(* Logix 5000 project; controller STAT 1756-L72 rev 20.12; software revision 20.04; part 31 of 34 *)
(* tags used below, declared in another part *)
   AUX_COND_KOELTOREN : REAL;
   AUX_LVL_KOEL : DINT;
   def_temp_iwts : BOOL;
   dmd_h2so4_ibt_ok : BOOL;
   ibtlancy1 : DINT;
   INT_COND_KOEL : integrat;
   INT_LVL_KOEL : integrat;
   L1_stat : DINT[20];
   L2_L3_OK : BOOL;
   L2_L3_ppas : DINT;
   L2_STAT : DINT[20];
   LVL_NITRIC : REAL;
   msg_W_lancy2 : MESSAGE;
   N : INT[255];
   naohL1VA4 : BOOL;
   naohL2VA4 : BOOL;
   op010 : DINT;
   real : REAL;
   S_BP_L2L3 : BOOL;
   S_COND_KOELTOREN : DINT;
   S_L2L3_Q_NAOH : DINT;
   S_LVL_KOELTOREN : DINT;
   S_LVL_nitric : REAL;
   S_STOCK_H2SO4 : DINT;
   S_STOCK_MAZ : DINT;
   S_STOCK_NAOH : DINT;
   S_T_CABINE_RED : DINT;
   S_T_in_CH_L3 : DINT;
   S_T_in_chaud_L123 : DINT;
   S_T_IWTS : DINT;
   S_T_OUT_CH_L3 : DINT;
   S_T_out_chaud_L123 : DINT;
   SCP_COND_KOELTOREN : SCP;
   SCP_LVL_KOELTOREN : SCP;
   SCP_lvl_nitric : SCP;
   scp_stck_acid : SCP;
   scp_stck_maz : SCP;
   scp_stck_soude : SCP;
   SCP_T_CABINE_L1 : SCP;
   scp_T_in_CH_L3 : SCP;
   scp_T_in_L12 : SCP;
   scp_T_iwts : SCP;
   scp_T_OUT_CH_L3 : SCP;
   scp_T_out_L12 : SCP;
   Seconde : BOOL;
   stat_L1 : DINT[20];
   stocklancy1 : DINT;
   stocklancy2 : DINT;
   stocklancy3 : DINT;
   stocklancy5 : DINT;   // alarme lvl 2 stock
   T1_cligno : TIMER;
   T_CABINE_RED : REAL;
   T_R_L2L3 : TIMER;
(* LANCY, continued *)

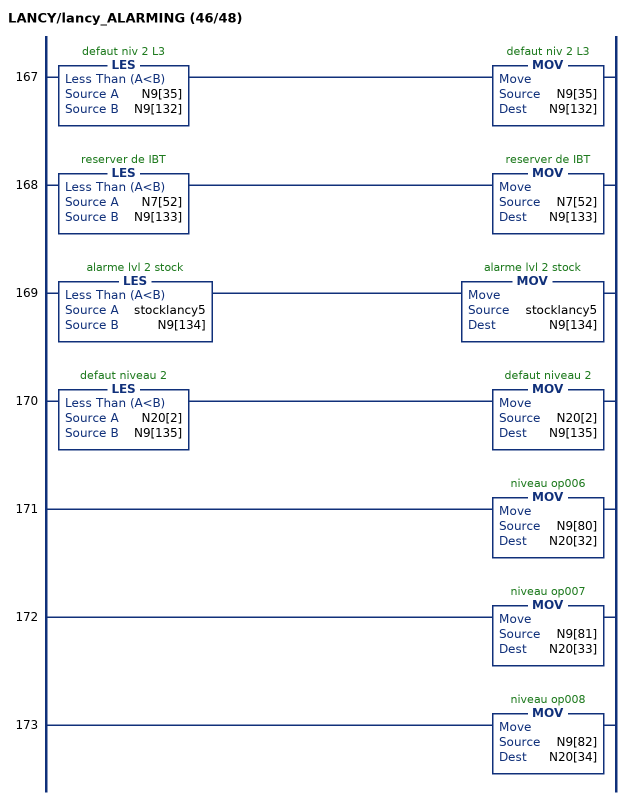
   [picture p626: LANCY/lancy_ALARMING rungs 167-173]
   167: LES(N9[35],N9[132])MOV(N9[35],N9[132]);
   168: LES(N7[52],N9[133])MOV(N7[52],N9[133]);
   169: LES(stocklancy5,N9[134])MOV(stocklancy5,N9[134]);
   170: LES(N20[2],N9[135])MOV(N20[2],N9[135]);
   171: MOV(N9[80],N20[32]);
   172: MOV(N9[81],N20[33]);
   173: MOV(N9[82],N20[34]);
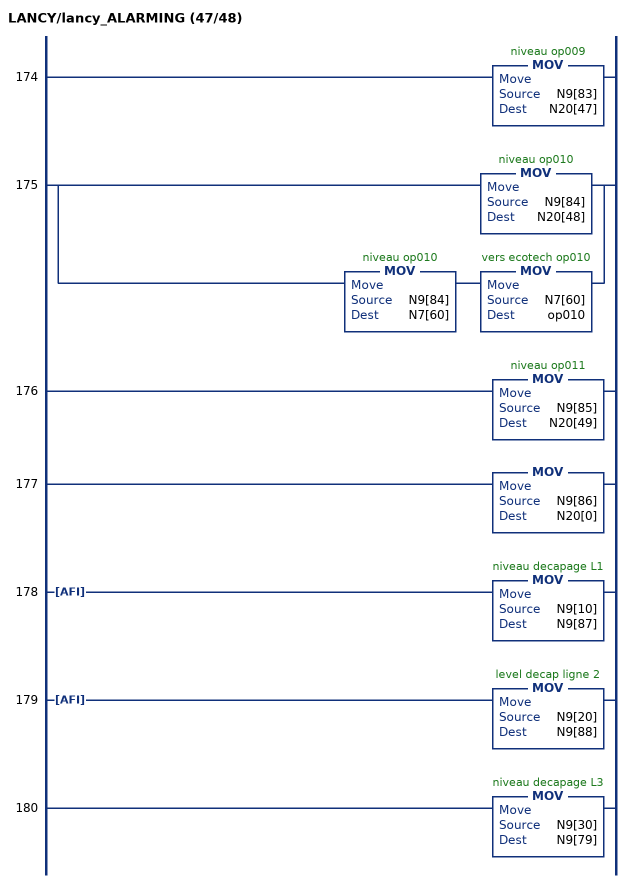
   174: MOV(N9[83],N20[47]);
   175: [MOV(N9[84],N20[48]) ,MOV(N9[84],N7[60]) MOV(N7[60],op010) ];
   176: MOV(N9[85],N20[49]);
   177: MOV(N9[86],N20[0]);
   178: AFI()MOV(N9[10],N9[87]);
   179: AFI()MOV(N9[20],N9[88]);
   180: MOV(N9[30],N9[79]);
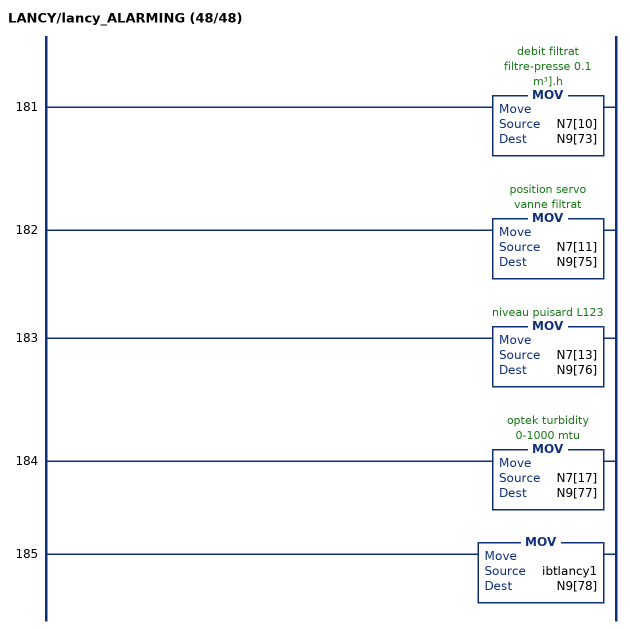
   181: MOV(N7[10],N9[73]);
   182: MOV(N7[11],N9[75]);
   183: MOV(N7[13],N9[76]);
   184: MOV(N7[17],N9[77]);
   185: MOV(ibtlancy1,N9[78]);
END_ROUTINE

ROUTINE lancy_apport_soude   (* ladder *)
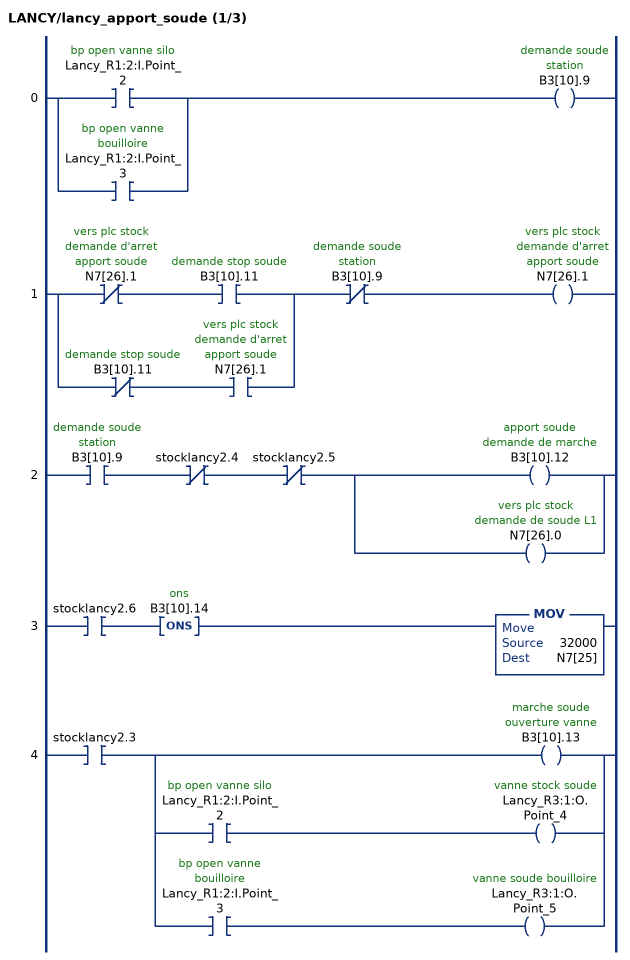
   0: [XIC(Lancy_R1:2:I.Point_2) ,XIC(Lancy_R1:2:I.Point_3) ]OTE(B3[10].9);
   1: [XIO(N7[26].1) XIC(B3[10].11) ,XIO(B3[10].11) XIC(N7[26].1) ]XIO(B3[10].9)OTE(N7[26].1);
   2: XIC(B3[10].9)XIO(stocklancy2.4)XIO(stocklancy2.5)[OTE(B3[10].12) ,OTE(N7[26].0) ];
   3: XIC(stocklancy2.6)ONS(B3[10].14)MOV(32000,N7[25]);
   4: XIC(stocklancy2.3)[OTE(B3[10].13) ,XIC(Lancy_R1:2:I.Point_2) OTE(Lancy_R3:1:O.Point_4) ,XIC(Lancy_R1:2:I.Point_3) OTE(Lancy_R3:1:O.Point_5) ];
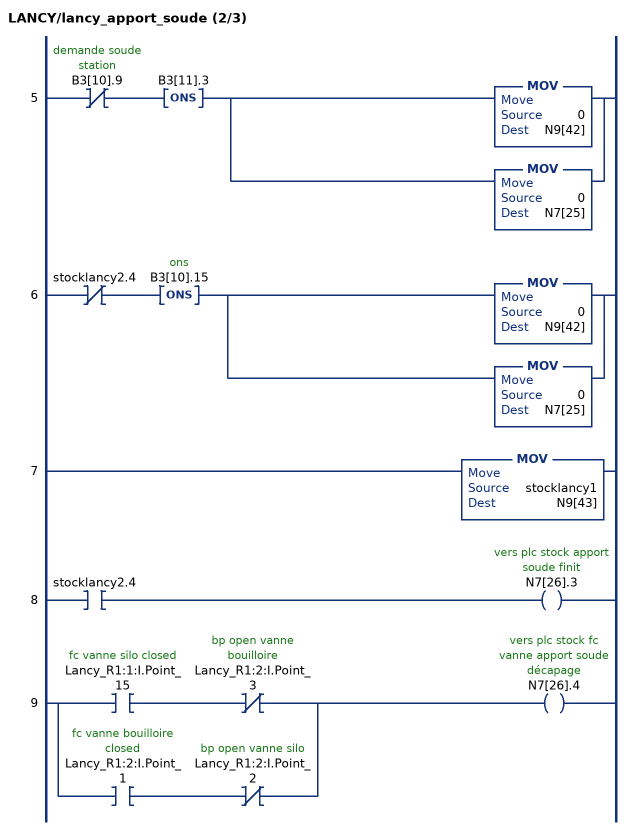
   5: XIO(B3[10].9)ONS(B3[11].3)[MOV(0,N9[42]) ,MOV(0,N7[25]) ];
   6: XIO(stocklancy2.4)ONS(B3[10].15)[MOV(0,N9[42]) ,MOV(0,N7[25]) ];
   7: MOV(stocklancy1,N9[43]);
   8: XIC(stocklancy2.4)OTE(N7[26].3);
   9: [XIC(Lancy_R1:1:I.Point_15) XIO(Lancy_R1:2:I.Point_3) ,XIC(Lancy_R1:2:I.Point_1) XIO(Lancy_R1:2:I.Point_2) ]OTE(N7[26].4);
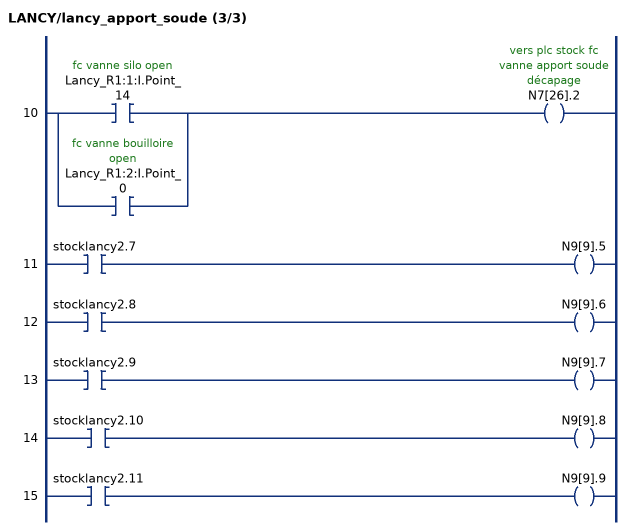
   10: [XIC(Lancy_R1:1:I.Point_14) ,XIC(Lancy_R1:2:I.Point_0) ]OTE(N7[26].2);
   11: XIC(stocklancy2.7)OTE(N9[9].5);
   12: XIC(stocklancy2.8)OTE(N9[9].6);
   13: XIC(stocklancy2.9)OTE(N9[9].7);
   14: XIC(stocklancy2.10)OTE(N9[9].8);
   15: XIC(stocklancy2.11)OTE(N9[9].9);
END_ROUTINE

ROUTINE NAOH   (* ladder *)
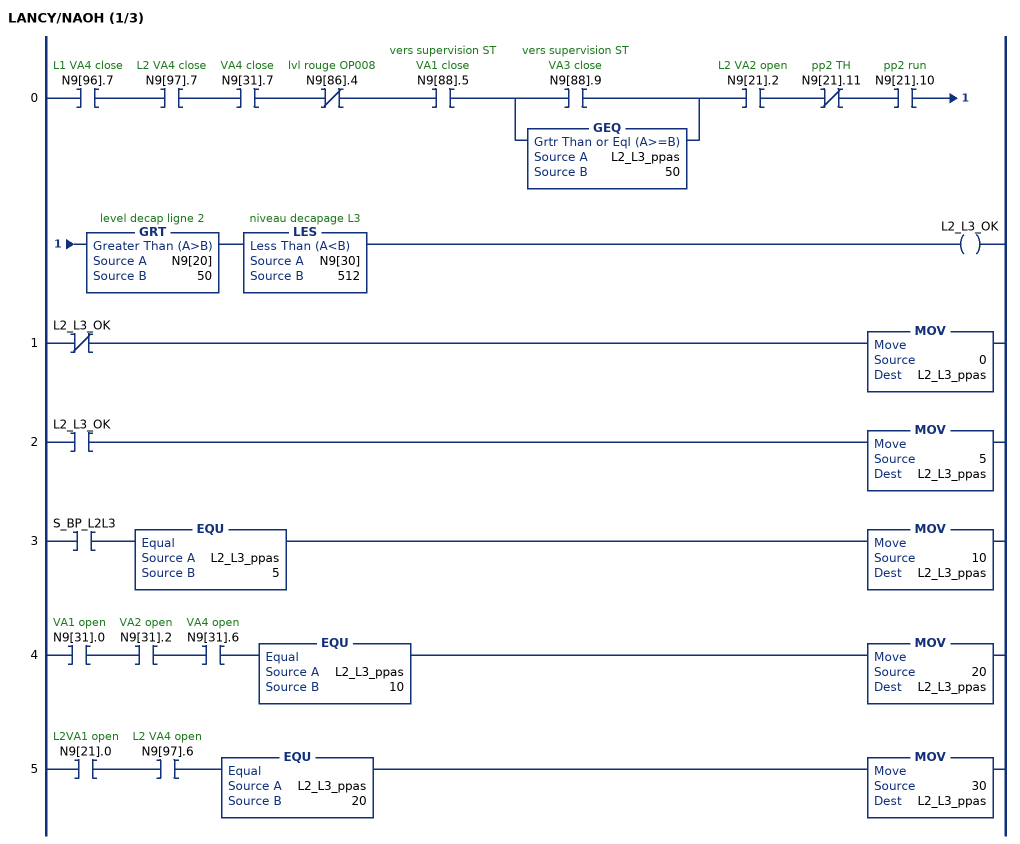
   0: XIC(N9[96].7)XIC(N9[97].7)XIC(N9[31].7)XIO(N9[86].4)XIC(N9[88].5)[XIC(N9[88].9) ,GEQ(L2_L3_ppas,50) ]XIC(N9[21].2)XIO(N9[21].11)XIC(N9[21].10)GRT(N9[20],50)LES(N9[30],512)OTE(L2_L3_OK);
   1: XIO(L2_L3_OK)MOV(0,L2_L3_ppas);
   2: XIC(L2_L3_OK)MOV(5,L2_L3_ppas);
   3: XIC(S_BP_L2L3)EQU(L2_L3_ppas,5)MOV(10,L2_L3_ppas);
   4: XIC(N9[31].0)XIC(N9[31].2)XIC(N9[31].6)EQU(L2_L3_ppas,10)MOV(20,L2_L3_ppas);
   5: XIC(N9[21].0)XIC(N9[97].6)EQU(L2_L3_ppas,20)MOV(30,L2_L3_ppas);
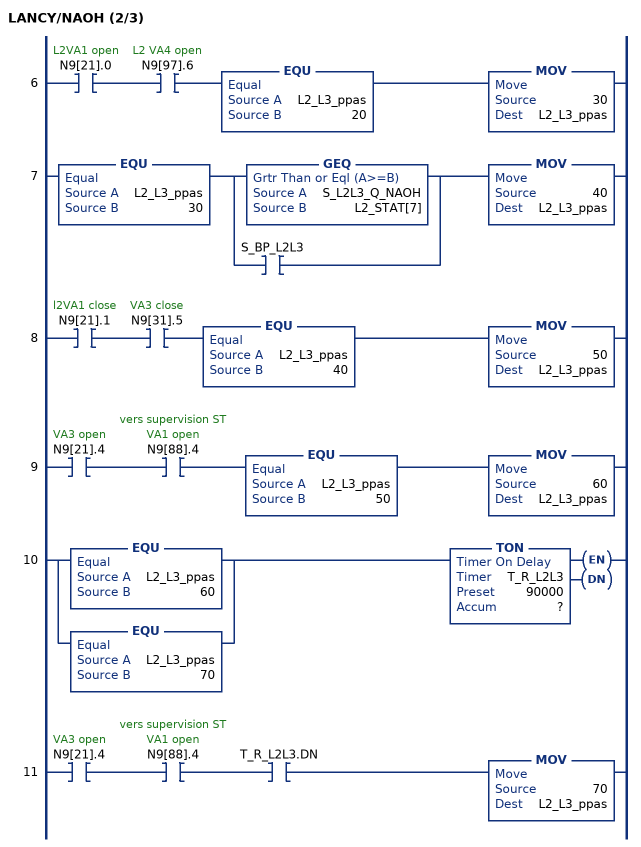
   6: XIC(N9[21].0)XIC(N9[97].6)EQU(L2_L3_ppas,20)MOV(30,L2_L3_ppas);
   7: EQU(L2_L3_ppas,30)[GEQ(S_L2L3_Q_NAOH,L2_STAT[7]) ,XIC(S_BP_L2L3) ]MOV(40,L2_L3_ppas);
   8: XIC(N9[21].1)XIC(N9[31].5)EQU(L2_L3_ppas,40)MOV(50,L2_L3_ppas);
   9: XIC(N9[21].4)XIC(N9[88].4)EQU(L2_L3_ppas,50)MOV(60,L2_L3_ppas);
   10: [EQU(L2_L3_ppas,60) ,EQU(L2_L3_ppas,70) ]TON(T_R_L2L3,?,?);
   11: XIC(N9[21].4)XIC(N9[88].4)XIC(T_R_L2L3.DN)MOV(70,L2_L3_ppas);
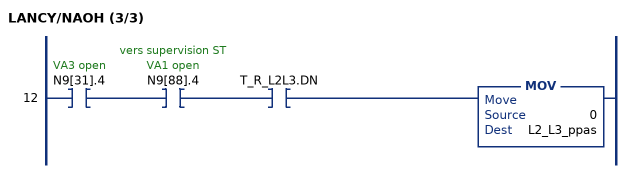
   12: XIC(N9[31].4)XIC(N9[88].4)XIC(T_R_L2L3.DN)MOV(0,L2_L3_ppas);
END_ROUTINE
END_PROGRAM

PROGRAM MainProgram
END_PROGRAM

PROGRAM stock   (* main routine MAIN_STOCK *)
VAR
   aa : DINT;
   B3 : DINT[50] := ([0] := 2#0000_0000_0000_0000_0000_1000_0010_0000, [2] := 2#0000_0000_0000_0000_0100_0010_1110_0000, [3] := 2#0000_0000_0000_0000_0000_0000_0000_0101, [5] := 2#0000_0000_0000_0000_0000_0000_1000_0000);
        [4].1   // L1 hs
        [4].2   // l2 hs
        [4].3   // l3 hs
        [0].0   // UNE VANNE SOUDE OUVERTE
        [0].4   // vanne acidedemarrage pompe
        [0].5   // one shot
        [0].6   // ons
        [0].7   // soude occupée
        [0].8   // soude déjaoccupé
        [0].9   // défautvanne soude
        [0].10   // ACIDE DEJAACCUPE
        [0].11   // ons
        [0].12   // acide occupe
        [0].14   // défautvanne acide
        [0].15   // AUX D2FAUTVANNE ACIDE
        [1].1   // ons
        [1].2   // apport soude
        [1].3   // acquit klaxonfuite acide
        [1].4   // acquit klaxonfuite soude
        [1].5   // acquit klaxonfuite mazout
        [1].6   // detectionfuiteacide
        [1].12   // apport acide
        [2].0   // ons
        [2].1   // ons
        [2].2   // ons
        [2].3   // ons
        [2].4   // ons
        [2].5   // ons
        [2].7   // ons
        [2].8   // ons
        [2].9   // ons
        [2].10   // ons
        [2].11   // ons
        [2].12   // ons
        [2].13   // ons
        [2].14   // ons
        [2].15   // ons
        [3].0   // fonctionnementdepuis supervision
        [3].1   // ARRET ENTRETIEN
        [3].2   // nouveau def
        [3].3   // rappel demandé
        [4].0   // stat hs
        [4].4   // l4 hs
        [5].7   // ons
   C5 : COUNTER[10];
   F8 : REAL[200] := ([2] := 863724.06, [3] := 863678.3, [5] := 24000.0, [7] := 1000.0, [10] := 17654.0, [11] := 20000.0, [12] := 9201.893, [13] := 48000.0, [14] := 24840.227, [15] := 45000.0, [16] := -750.11444, [17] := -750.11444, [18] := 2135.205, [19] := 2142.53, [20] := 2033.7975, [21] := 1750.6666, [22] := 2993.7632, [23] := 150.19885, [25] := 44558.395, [26] := 80344.15, [27] := 2182.817, [29] := 281.0, [30] := 24832.748, [31] := -3.7382812, [32] := 17654.0, [34] := 9201.893, [35] := -3.8154297, [36] := 5102.8765, [37] := 2410.5056, [38] := 7013.7407, [41] := 0.6, [42] := 50.0, [43] := 50.000046, [46] := -863724.06, [47] := 50.0, [48] := 50.000046, [50] := 318801.06, [52] := -318801.06, [61] := 1750.6666, [62] := 2993.7632, [63] := 150.19885);
        [2]   // 0.2 L].pulsetotalacide
        [3]   // memo acidepassé
        [4]   // quantitédernièreenvoi acide
        [10]   // Stock acide
        [12]   // stock mazout
        [14]   // stock soude
        [16]   // temperature entréeChaudière Ligne 1-2
        [17]   // temperature desortie chaudièreLigne 1-2
        [18]   // temp entréechaudierecolmatage L3
        [19]   // temp sortiechaudierecolmatage L3
        [20]   // total soudevers station
        [21]   // total soudevers L1
        [22]   // total soudevers L2
        [23]   // total soudevers L3
        [24]   // total soudevers L4
        [25]   // total soudevers L2
        [26]   // total soudevers L1
        [27]   // chaudiere iwts
        [30]   // NIVEAU PRECEDENTSOUDE
        [31]   // PERTE SOUDE SUR UNEMINUTE
        [32]   // PERTE ACIDE SUR UNEMIN
        [33]   // MEMO NIVEAI ACIDE1 MIN AVANT
        [34]   // MEMO MAZOUT 1 MIN
        [35]   // PERTE MAZOUT SUR1 MIN
        [36]   // totalacideL1
        [37]   // totalacideL2
        [38]   // totalacideL3
        [39]   // totalacideL4
        [40]   // quantité demandéedepuis ligne
        [41]   // quantité soudepassée
        [42]   // quantité acidedemandéedepuis ligne
        [43]   // quantité acidepassée
        [45]   // aux total acide
        [46]   // aux total acide
        [47]   // aux total acide
        [48]   // quantité acidepassé
        [50]   // total soudepassée en L
        [62]   // MEMO FLOW TO L2
        [63]   // MEMO FLOW TO L3
   I1 : DINT;
   I1_000_Bit00 : ALIAS FOR stock:1:I.Point_0;   // disjoncteur algemeen
   I1_000_Bit01 : ALIAS FOR stock:1:I.Point_1;   // alim rechauffeur1
   I1_000_Bit02 : ALIAS FOR stock:1:I.Point_2;   // alim rechauffeur2
   I1_000_Bit03 : ALIAS FOR stock:1:I.Point_3;   // alim rechauffeur 3
   I1_000_Bit04 : ALIAS FOR stock:1:I.Point_4;   // alim rechauffeur 4
   I1_000_Bit05 : ALIAS FOR stock:1:I.Point_5;   // alim rechauffeur 5
   I1_000_Bit06 : ALIAS FOR stock:1:I.Point_6;   // protection pompesoude
   I1_000_Bit07 : ALIAS FOR stock:1:I.Point_7;   // protection pmp 2 acide
   I1_000_Bit08 : ALIAS FOR stock:1:I.Point_8;   // protection pmp acide
   I1_000_Bit09 : ALIAS FOR stock:1:I.Point_9;
   I1_000_Bit10 : ALIAS FOR stock:1:I.Point_10;
   I1_000_Bit11 : ALIAS FOR stock:1:I.Point_11;
   I1_000_Bit12 : ALIAS FOR stock:1:I.Point_12;
   I1_000_Bit15 : ALIAS FOR stock:1:I.Point_15;   // arret urgence
   I1_001_Bit01 : ALIAS FOR stock:1:I.Point_17;   // reset arret urgence
   I1_001_Bit02 : ALIAS FOR stock:1:I.Point_18;   // start pompe soude
   I1_001_Bit03 : ALIAS FOR stock:1:I.Point_19;   // stop pompe soude
   I1_001_Bit04 : ALIAS FOR stock:1:I.Point_20;   // start pompe acide
   I1_001_Bit05 : ALIAS FOR stock:1:I.Point_21;   // stop pompe acide
   I1_001_Bit08 : ALIAS FOR stock:1:I.Point_24;   // local ]. distance
   I1_001_Bit09 : ALIAS FOR stock:1:I.Point_25;   // select.pmp soude sur drive
   I1_001_Bit10 : ALIAS FOR stock:1:I.Point_26;   // select.pmp soude sur ultima
   I1_001_Bit11 : ALIAS FOR stock:1:I.Point_27;   // fault drivepmp soude
   I2 : DINT;
   I2_000_Bit00 : ALIAS FOR stock:2:I.Point_0;   // detection fuite soud
   I2_000_Bit01 : ALIAS FOR stock:2:I.Point_1;   // detection fuite acid
   I2_000_Bit02 : ALIAS FOR stock:2:I.Point_2;   // detection fuite mazo
   I2_000_Bit03 : ALIAS FOR stock:2:I.Point_3;   // wegskraan soude open
   I2_000_Bit04 : ALIAS FOR stock:2:I.Point_4;   // wegskraan soude dich
   I2_000_Bit05 : ALIAS FOR stock:2:I.Point_5;   // start pompe acidedepuis ligne
   I2_000_Bit06 : ALIAS FOR stock:2:I.Point_6;   // start pompe acidedepuis ligne RESERVE
   I2_000_Bit07 : ALIAS FOR stock:2:I.Point_7;   // overfill stockagesoude
   I2_000_Bit08 : ALIAS FOR stock:2:I.Point_8;   // detection acideencuvement
   I2_000_Bit09 : ALIAS FOR stock:2:I.Point_9;   // detection soudeencuvement
   I2_000_Bit10 : ALIAS FOR stock:2:I.Point_10;   // fv vannesecuriteacide OUVERT
   I2_000_Bit11 : ALIAS FOR stock:2:I.Point_11;   // fv vannesecuriteacide FERME
   I2_000_Bit12 : ALIAS FOR stock:2:I.Point_12;   // chaudière wanson0= on 1= off
   I2_000_Bit13 : ALIAS FOR stock:2:I.Point_13;   // chaudière colmatageLigne 30= on 1= off
   I2_000_Bit14 : ALIAS FOR stock:2:I.Point_14;   // DEFAUT CHAUDIEREiwts
   I2_001_Bit00 : ALIAS FOR stock:2:I.Point_16;   // NAOHL1 VA4FC O
   I2_001_Bit01 : ALIAS FOR stock:2:I.Point_17;   // NAOHL1 VA4FC F
   I2_001_Bit02 : ALIAS FOR stock:2:I.Point_18;   // NAOHL2 VA4FC O
   I2_001_Bit03 : ALIAS FOR stock:2:I.Point_19;   // NAOHL2 VA4FC O
   I2_001_Bit06 : ALIAS FOR stock:2:I.Point_22;   // pulse debitmetreacide 0.2 l
   I2_001_Bit07 : ALIAS FOR stock:2:I.Point_23;   // pulse eau in tourL1 &2
   I2_001_Bit15 : ALIAS FOR stock:2:I.Point_31;   // pulse 0.1L passé
   I4 : AB:1746_NI8_C63AF0D1:I:0;
   I4_001 : ALIAS FOR stock:4:I.Channel_1_Data;   // level soude
   I4_002 : ALIAS FOR stock:4:I.Channel_2_Data;   // level acide
   I4_003 : ALIAS FOR stock:4:I.Channel_3_Data;   // level mazout
   I4_004 : ALIAS FOR stock:4:I.Channel_4_Data;
   I4_005 : ALIAS FOR stock:4:I.Channel_5_Data;
   I4_006 : ALIAS FOR stock:4:I.Channel_6_Data;
   I4_007 : ALIAS FOR stock:4:I.Channel_7_Data;
   I5 : INT[8] := ([0] := 2#0000_1100_1100_1101, [1] := 2#0001_0000_0011_0101, [2] := 2#0011_0111_1011_0100, [3] := 2#0001_0001_1111_1000, [4] := 2#0000_1100_1101_0101, [5] := 2#0001_1000_1001_0100);
   I5_000 : ALIAS FOR stock:5:I.Channel_0_Data;
   I5_001 : ALIAS FOR stock:5:I.Channel_1_Data;
   I5_002 : ALIAS FOR stock:5:I.Channel_2_Data;
   I5_003 : ALIAS FOR stock:5:I.Channel_3_Data;
   I5_004 : ALIAS FOR stock:5:I.Channel_4_Data;
   I5_005 : ALIAS FOR stock:5:I.Channel_5_Data;
   N20 : DINT[100] := ([1] := 8, [2] := 3, [5] := 3, [10] := 2, [20] := 64, [21] := 61967, [25] := 64, [30] := 10, [31] := 1);
        [1]   // DEFAUT PRIORITE 1
        [2]   // DEFAUT PRIORITE 2
        [5].0   // DEFAULT
        [5].1   // NEW DEFAULT
        [9].1   // ack STOCK
        [10].0   // chaudiere wanson on
        [10].1   // chaudière colmatageLigne 3 on
        [20].0   // defautdisjoncteur algemeen
        [20].1   // DEFAUTalim rechauffeur1
        [20].2   // DEFAUTalim rechauffeur2
        [20].3   // DEFAUTalim rechauffeur 3
        [20].4   // DEFAUTalim rechauffeur 4
        [20].5   // DEFAUTalim rechauffeur 5
        [20].6   // DEFAUTprotection pompesoude
        [20].7   // DEFAUTprotection pmpmazout
        [20].8   // DEFAUTprotection pmp acide
        [20].9   // DEFAUTarret urgence
        [20].10   // DEFAUTdetection fuite soud
        [20].11   // DEFAUTdetection fuite acid
        [20].12   // DEFAUTdetection fuite mazo
        [20].13   // DEFAUToverfill stockagesoude
        [20].14   // DEFAUTdetection acideencuvement
        [20].15   // DEFAUTdetection soudeencuvement
        [21].0   // DEFAUTPOSITION VANNEL1 VA4
        [21].1   // DEFAUTPOSITION VANNEL2 VA4
        [21].2   // DEFAUTPOSITION VANNESOUDE VERS LIGNES
        [21].3   // DEFAUTPOSITION VANNEACIDE VERS LIGNES
        [21].4   // DEFAUT FLOW SOUDE
        [21].5   // DEFAUT NIVEAU SOUDEHH
        [21].6   // DEFAUT NIVEAU SOUDELL
        [21].7   // DEFAUT FILL OUTNOAH TANK
        [21].8   // DEFAUT NIVEAU ACIDEHH
        [21].9   // DEFAUT NIVEAU ACIDELL
        [21].10   // DEFAUT FILL OUTH2SO4 TANK
        [21].11   // DEFAUT NIVEAU MAZOUTHH
        [21].12   // DEFAUT NIVEAU MAZOUTLL
        [21].13   // DEFAUT FILL OUTMAZOUT TANK
        [21].14   // DEFAUT CHAUDIEREiwts
        [21].15   // defautchaudierecolmatage L3
        [25].0   // defautdisjoncteur algemeen
        [25].1   // DEFAUTalim rechauffeur1
        [25].2   // DEFAUTalim rechauffeur2
        [25].3   // DEFAUTalim rechauffeur 3
        [25].4   // DEFAUTalim rechauffeur 4
        [25].5   // DEFAUTalim rechauffeur 5
        [25].6   // DEFAUTprotection pompesoude
        [25].7   // DEFAUTprotection pmpmazout
        [25].8   // DEFAUTprotection pmp acide
        [25].9   // DEFAUTarret urgence
        [25].10   // DEFAUTdetection fuite soud
        [25].11   // DEFAUTdetection fuite acid
        [25].12   // DEFAUTdetection fuite mazo
        [25].13   // overfill stockagesoude
        [25].14   // DEFAUTdetection acideencuvement
        [25].15   // DEFAUTdetection soudeencuvement
        [26].0   // DEFAUTPOSITION VANNEL1 VA4
        [26].1   // DEFAUTPOSITION VANNEL2 VA4
        [26].2   // DEFAUTPOSITION VANNESOUDE VERS LIGNES
        [26].3   // DEFAUTPOSITION VANNEACIDE VERS LIGNES
        [26].4   // DEFAUT FLOW SOUDE
        [26].5   // DEFAUT NIVEAU SOUDEHH
        [26].6   // DEFAUT NIVEAU SOUDELL
        [26].7   // DEFAUT FILL OUTNOAH TANK
        [26].8   // DEFAUT NIVEAU ACIDEHH
        [26].9   // DEFAUT NIVEAU ACIDELL
        [26].10   // DEFAUT FILL OUTH2SO4 TANK
        [26].11   // DEFAUT NIVEAU MAZOUTHH
        [26].12   // DEFAUT NIVEAU MAZOUTLL
        [26].13   // DEFAUT FILL OUTMAZOUT TANK
        [26].14   // DEFAUT CHAUDIEREiwts
        [26].15   // memo defautchaudierecolmatage L3
        [30]   // NOMBRE DE DEFAUTS
        [31]   // MEMONOMBRE DE DEFAUTS
   N7 : DINT[255] := ([1] := 131701, [3] := 3850, [4] := 3800, [10] := 21, [15] := 281, [18] := 314857, [20] := 10, [21] := -4, [66] := -32752, [68] := 336, [88] := 50, [108] := 80, [126] := 3488, [127] := 35200, [166] := 3488, [167] := 35200, [206] := 3488, [207] := 35200, [246] := 3488);
        [1]   // gxf
        [2]   // flow acide
        [10].0   // stock acide pas haut
        [10].1   // stock acide pas bas
        [10].2   // stock mazout pashaut
        [10].3   // stock mazout pas bas
        [10].4   // stock soude L1 pashaut
        [10].5   // stock soude L1 pasbas
        [10].7   // stock soude L2 pasbas
        [10].8   // stock soude L3 pashaut
        [10].9   // stock soude L3 pasbas
        [10].10   // PVvanne soude L1fermée
        [10].13   // de PVchargement en cours
        [10].14   // DE PVBP EV SOUDE L1
        [11].0   // DE PVBP EV SOUDE L3
        [11].1   // vers PVfuite stock acide
        [11].2   // vers PVfuite stock mazout
        [11].3   // fuite soude
        [15]   // T° ambiantecabine RED L1
        [16]   // conductivité en µS
        [17]   // niveau eautour refroidissement
        [18]   // total eau tour L1 2
        [20].0   // NAOHL1 VA4FC O
        [20].1   // NAOHL1 VA4FC F
        [20].2   // NAOHL2 VA4FC O
        [20].3   // NAOHL2 VA4FC F
        [30]   // MESSAGE TO LANCY
        [46].2   // DE PLC 1VANNE SOUDEL1 OUVERTE
        [50]   // communication avecplc L1 read
        [65]   // quantité soudedemandée L1
        [66].0   // DE PLC L1demande soudeL1
        [66].1   // DE PLC L1demandearret soude L1
        [66].2   // de plc ligne 1fc vanne soudeouverte
        [66].3   // de plc ligne 1apport soudefinit
        [66].4   // de plc ligne 1fc vanne soudefermée
        [66].15   // de line 1line 1 run
        [67]   // quantité acidedemandée L1
        [68].0   // DE PLC L1demande acide
        [68].1   // DE PLC L1demandearret acide L1
        [68].2   // de plc ligne 1fc vanne acideano ouv
        [68].3   // de plc ligne 1apport acidefinit
        [68].4   // de plc ligne 1fc vanne acideano ferme
        [68].5   // de plc ligne 1fc vanne acideneut ouv
        [68].6   // de plc ligne 1fc vanne acideneut ferme
        [68].7   // de plc ligne 1fc vanne acidecolo ouv
        [68].8   // de plc ligne 1fc vanne acidecolo fermé
        [70]   // communication avecplc L1 write
        [85]   // quantité souderestante L1
        [86].0   // vers plc l1 fuiteacide
        [86].1   // vers plc l1fuite soude
        [86].2   // vers plc L1fuite mazout
        [86].3   // vers plc L1ouvrir vannesoude
        [86].4   // vers plc L1apport soudefinit L1
        [86].5   // vers plc L1apport soudeoccupé
        [86].6   // vers plc L1apport soudeL1 accordé
        [86].7   // VERS PLC L1SOUDE VERS L1
        [86].8   // VERS PLC L1SOUDE VERS L2
        [86].9   // VERS PLC L1SOUDE VERS L3
        [86].10   // VERS PLC L1SOUDE VERS L4
        [86].11   // VERS PLC L1SOUDE VERS STAT
        [86].12   // DEFAULT FLOW TO L1VERS SLC
        [87]   // vers plc L1
        [87].3   // vers plc L1ouvrir vanneacide
        [87].4   // vers plc L1apport acidefinit L1
        [87].5   // vers plc L1apport acideoccupé
        [87].6   // vers plc L1apport acideaccordé
        [87].7   // VERS PLC L1acide VERS ano L1
        [87].8   // VERS PLC L1acideVERS L2
        [87].9   // VERS PLC L1acide VERS L3
        [87].10   // VERS PLC L1acide VERS L4
        [87].11   // VERS PLC L1acide VERS neutralL1
        [87].12   // VERS PLC L1 acideneutralL2
        [87].13   // VERS PLC L1acide neutralL3
        [87].14   // VERS PLC L1 acide VEL4
        [88]   // quantité aciderestante L1
        [90]   // communication avecplc L2 read
        [105]   // quantité soudedemandée L2
        [106].0   // DE PLC L2demande soudeL2
        [106].1   // DE PLC L2demandearret soude
        [106].2   // de plc ligne 2fc vanne soudeouverte
        [106].4   // de plc ligne 2fc vanne soudefermée
        [106].15   // de line 2line 2 run
        [107]   // quantité acidedemandée L2
        [108].0   // DE PLC L2demande acide
        [108].1   // DE PLC L2demandearret acide L2
        [108].2   // de plc ligne 2fc vanne acideouverte
        [108].4   // de plc ligne 2fc vanne acidefermée
        [108].5   // de plc ligne 2fc vanne acideneutral ouv
        [108].6   // de plc ligne 2fc vanne acideneutral ferm
        [110]   // communication avecplc L2 write
        [125]   // quantité souderestante L2
        [126].3   // vers plc L2ouvrir vannesoude
        [126].4   // vers plc L2apport soudefinit L2
        [126].5   // vers plc L2apport soudeoccupé
        [126].6   // vers plc L2apport soudeL2 accordé
        [126].7   // VERS PLC L2SOUDE VERS L1
        [126].8   // VERS PLC L2SOUDE VERS L2
        [126].9   // VERS PLC L2SOUDE VERS L3
        [126].10   // VERS PLC L2SOUDE VERS L4
        [126].11   // VERS PLC L2SOUDE VERS STAT
        [126].12   // DEFAULT FLOW TO L2VERS SLC
        [127].3   // vers plc L2ouvrir vanneacide
        [127].4   // vers plc L2apport acidefinit L2
        [127].5   // vers plc L2apport acideoccupé
        [127].6   // vers plc L2apport acideaccordé
        [127].7   // VERS PLC L2acide VERS ano L1
        [127].8   // VERS PLC L2acide VERS L2
        [127].9   // VERS PLC L2acide VERS L3
        [127].10   // VERS PLC L2acide VERS L4
        [127].11   // VERS PLC L2acide VERS neutralL1
        [127].12   // VERS PLC L2 acideneutralL2
        [127].13   // VERS PLC L2 acideneutralL3
        [127].14   // VERS PLC L2 acide VEL4
        [128]   // quantite acidepassé l2
        [130]   // communication L3read
        [139]   // MEMODEFAUT DEGRAISSAGE
        [145]   // quantité soudedemandéel3
        [146].0   // DE PLC L3demande soudeL3
        [146].1   // DE PLC L3demandearret soude L3
        [146].2   // de plc ligne 3fc vanne soudeouverte
        [146].4   // de plc ligne 3fc vanne soudefermée
        [146].15   // ligne 3 runcolmatage
        [147]   // quantité acidedemandée l3
        [148].0   // DE PLC L3demande acide L3
        [148].1   // DE PLC L3demandearret acide L3
        [148].2   // de plc ligne 3fc vanneacide ouverte
        [148].4   // de plc ligne 3fc vanne acidefermée
        [148].5   // de plc ligne 3fc vanneacide neutral ouv
        [148].6   // de plc ligne 3fc vanneacide neutral ferm
        [150]   // communication L3write
        [165]   // quantité souderestante L3
        [166].3   // vers plc L3ouvrir vannesoude
        [166].4   // vers plc L3apport soudeL3 finit
        [166].5   // vers plc L3apport soudeoccupé
        [166].6   // vers plc L3apport soudeL3 accordé
        [166].7   // VERS PLC L3SOUDE VERS L1
        [166].8   // VERS PLC L3SOUDE VERS L2
        [166].9   // VERS PLC L3SOUDE VERS L3
        [166].10   // VERS PLC L3SOUDE VERS L4
        [166].11   // VERS PLC L3SOUDE VERS STAT
        [166].12   // DEFAULT FLOW TO L3VERS SLC
        [167].3   // vers plc L3ouvrir vanneacide
        [167].4   // vers plc L3apport acidefinit L3
        [167].5   // apport acide occupé
        [167].6   // apport acide accordé
        [167].7   // VERS PLC L3acide VERS ano L1
        [167].8   // VERS PLC L3acide VERS L2
        [167].9   // VERS PLC L3acide VERS L3
        [167].10   // VERS PLC L4acide VERS L4
        [167].11   // VERS PLC L3acide VERS neutralL1
        [167].12   // VERS PLC L3 acideneutralL2
        [167].13   // VERS PLC L3acideneutral L3
        [167].14   // VERS PLC L3 acide VEL4
        [168]   // quantite acidepassé l3
        [170]   // communicationL4
        [185]   // quantité soudedemandéel4
        [186].0   // DE PLC L4demande soudeL4
        [186].1   // DE PLC L4demandearret soude l4
        [186].2   // de plc ligne 4fc vanne soudeouverte
        [186].4   // de plc ligne 4fc vanne soudefermée
        [187]   // quantité acidedemandée L4
        [188].0   // DE PLC L4demande acide
        [188].1   // DE PLC L4demandearret acide L4
        [188].2   // de plc ligne 4fc vanne acideouverte
        [188].4   // de plc ligne 3fc vanne acidefermée
        [188].5   // de plc ligne 4fc vanne acideneutral ouv
        [188].6   // de plc ligne 4fc vanne acideneutral ferme
        [190]   // communicationL4
        [205]   // quantité souderestante L4
        [206].3   // vers plc L4ouvrir vannesoude
        [206].4   // vers plc L4apport soudeL4 finit
        [206].5   // vers plc L4apport soudeoccupé
        [206].6   // vers plc L4apport soudeL4 accordé
        [206].7   // VERS PLC L4SOUDE VERS L1
        [206].8   // VERS PLC L4SOUDE VERS L2
        [206].9   // VERS PLC L4SOUDE VERS L3
        [206].10   // VERS PLC L4SOUDE VERS L4
        [206].11   // VERS PLC L4SOUDE VERS STAT
        [207].3   // vers plc L4ouvrir vanneacide
        [207].4   // vers plc L4apport acidefinit L4
        [207].5   // vers plc L4apport acideoccupé
        [207].6   // vers plc L4apport acideaccordé
        [207].7   // VERS PLC L4acide VERS ano L1
        [207].8   // VERS PLC L4acide VERS L2
        [207].9   // VERS PLC L4acide VERS L3
        [207].10   // VERS PLC L4acide VERS L4
        [207].11   // VERS PLC L4acide VERS neutralL1
        [207].12   // VERS PLC L4 acideneutralL2
        [207].13   // VERS PLC L4acide neutralL3
        [207].14   // VERS PLC L4 acide VEL4
        [208]   // quantite acidepassé l4
        [210]   // lancy
        [226].0   // DE PLC statdemande soudestation
        [226].1   // DE PLC statdemandearret soude stat
        [226].2   // de plc ligne STATfc vanne soudeouverte
        [226].4   // de plc stationfc vanne soudefermée
        [230]   // lancy
        [245]   // quantité souderestante station
        [246].3   // vers plc statouvrir vannesoude
        [246].4   // vers plc statapport soudestat finit
        [246].5   // vers plc statapport soudeoccupé
        [246].6   // vers plc statapport soudestat accordé
        [246].7   // VERS PLC STATSOUDE VERS L1
        [246].8   // VERS PLC STATSOUDE VERS L2
        [246].9   // VERS PLC L1SOUDE VERS STAT
        [246].10   // VERS PLC STATSOUDE VERS L4
        [246].11   // VERS PLC STATSOUDE VERS STAT
   N9 : DINT[1] := ([0] := 10);
        [0].0   // vers supervNAOHL1 VA4 FC O
        [0].1   // vers superv NAOHL1 VA4FC F
        [0].2   // vers superv NAOHL2 VA4FC O
        [0].3   // vers superv NAOHL2 VA4FC F
   nitric_occupe : BOOL := 1;
   O3 : INT[2];
   O3_000_Bit00 : ALIAS FOR stock:3:O.Point_0;   // pompe soude
   O3_000_Bit01 : ALIAS FOR stock:3:O.Point_1;   // lampe bp start pmp s
   O3_000_Bit02 : ALIAS FOR stock:3:O.Point_2;   // pompe acide
   O3_000_Bit03 : ALIAS FOR stock:3:O.Point_3;   // L BP start pmp acide
   O3_000_Bit04 : ALIAS FOR stock:3:O.Point_4;   // pompe acide 2
   O3_000_Bit05 : ALIAS FOR stock:3:O.Point_5;   // L bp start pmp acide
   O3_000_Bit06 : ALIAS FOR stock:3:O.Point_6;   // lampe BP sur ligne p
   O3_000_Bit07 : ALIAS FOR stock:3:O.Point_7;
   O3_000_Bit08 : ALIAS FOR stock:3:O.Point_8;   // vanne soude
   O3_000_Bit09 : ALIAS FOR stock:3:O.Point_9;   // vannesecuriteacide
   O3_000_Bit11 : ALIAS FOR stock:3:O.Point_11;   // pompe adeokkoeltoren L1-2
   O3_000_Bit12 : ALIAS FOR stock:3:O.Point_12;   // remplissage tourrefroidissement
   O3_000_Bit13 : ALIAS FOR stock:3:O.Point_13;   // spuyvidange tour
   O3_000_Bit14 : ALIAS FOR stock:3:O.Point_14;   // power drivepmp soude
   O3_000_Bit15 : ALIAS FOR stock:3:O.Point_15;   // run drivepmp soude
   O3_001_Bit00 : ALIAS FOR stock:3:O.Point_16;   // L storing pmp soude
   O3_001_Bit01 : ALIAS FOR stock:3:O.Point_17;   // L storing pmp acide
   O3_001_Bit02 : ALIAS FOR stock:3:O.Point_18;   // l storing pmp mazout
   O3_001_Bit03 : ALIAS FOR stock:3:O.Point_19;   // L arret urgence
   O3_001_Bit04 : ALIAS FOR stock:3:O.Point_20;   // feu rouge trop plein
   O3_001_Bit05 : ALIAS FOR stock:3:O.Point_21;   // klaxon plein soude
   O3_001_Bit06 : ALIAS FOR stock:3:O.Point_22;   // feu rouge acide
   O3_001_Bit07 : ALIAS FOR stock:3:O.Point_23;   // klaxon trop plein ac
   O3_001_Bit08 : ALIAS FOR stock:3:O.Point_24;   // feu rouge trop plein
   O3_001_Bit09 : ALIAS FOR stock:3:O.Point_25;   // klaxon trop pleinmazout
   O3_001_Bit10 : ALIAS FOR stock:3:O.Point_26;   // reset arret urgence
   O3_001_Bit11 : ALIAS FOR stock:3:O.Point_27;   // L1 VA4
   O3_001_Bit12 : ALIAS FOR stock:3:O.Point_28;   // NAOHL2 VA4
   O3_001_Bit14 : ALIAS FOR stock:3:O.Point_30;   // drive pmp soudeV1
   O3_001_Bit15 : ALIAS FOR stock:3:O.Point_31;   // drive pmp soudeV2
   O4 : INT[8];
   O5 : INT[8];
   ons11 : BOOL;
   PMP_SOUDE : BOOL;
   R6 : CONTROL[10];
   S : INT[164];
   S24 : ALIAS FOR S[24];
   S_bp_dmd_naoh : BOOL;
   s_def_pmp_h2so4 : BOOL := 1;
   s_def_pmp_naoh : BOOL := 1;
   s_fc_v_h2so4_ferm : BOOL := 1;
   s_fc_v_h2so4_ouv : BOOL;
   S_ok_pmp_nitrique : BOOL := 1;
   S_pmp2_h2so4 : BOOL;
   s_pmp_h2so4 : BOOL;
   S_pmp_naoh : BOOL := 1;
   S_run_pmp_nitrique : BOOL;
   S_V_NAOH : BOOL;
   T4 : TIMER[50] := ([3].PRE := 18000000, [4].EN := 1, [4].DN := 1, [10].TT := 1, [10].DN := 1, [15].PRE := 5000, [15].ACC := 100, [15].EN := 1, [15].TT := 1, [21].EN := 1, [21].TT := 1, [22].ACC := 50, [22].EN := 1, [22].DN := 1, [23].ACC := 50, [23].EN := 1, [23].DN := 1, [24].ACC := 50, [25].PRE := 7200000, [25].ACC := 1693300, [25].EN := 1, [25].TT := 1, [26].PRE := 240000, [26].ACC := 240000, [27].EN := 1, [27].DN := 1, [28].ACC := 50);
        [1]   // tempo recouvrementcom.
        [2]   // stabilisationdemande
        [3]   // pompe acidearretée
        [5]   // DEFAULT FLOW TO L1
        [6]   // DEFAULT FLOW TO L2
        [7]   // DEFAULT FLOW TO L3
        [8]   // DEFAULT FLOW TO L4
        [9]   // presence defautnon acquité
        [10]   // envoi rappeldefautnon acquité
        [11]   // tempo recouvrementcom
        [12]   // stabilisation demandacide
        [14]   // vanne acideouverte
        [15]   // tempo cycle decommunication
        [16]   // POSITION VANNEL1 VA4
        [17]   // DEFAUTPOSITION VANNEL2 VA4
        [18]   // DEFAUTPOSITION VANNESOUDE VERS LIGNES
        [19]   // DEFAUTPOSITION VANNEACIDE VERS LIGNES
        [20]   // DEFAUT FLOW SOUDE
        [21]   // TEMPO 1 MIN
        [23]   // temp hyteresis
        [27]   // tof fermeture vannesoude
        [28]   // tof ouverture vannesoude
END_VAR

ROUTINE _6_KOELTOEREN   (* ladder *)
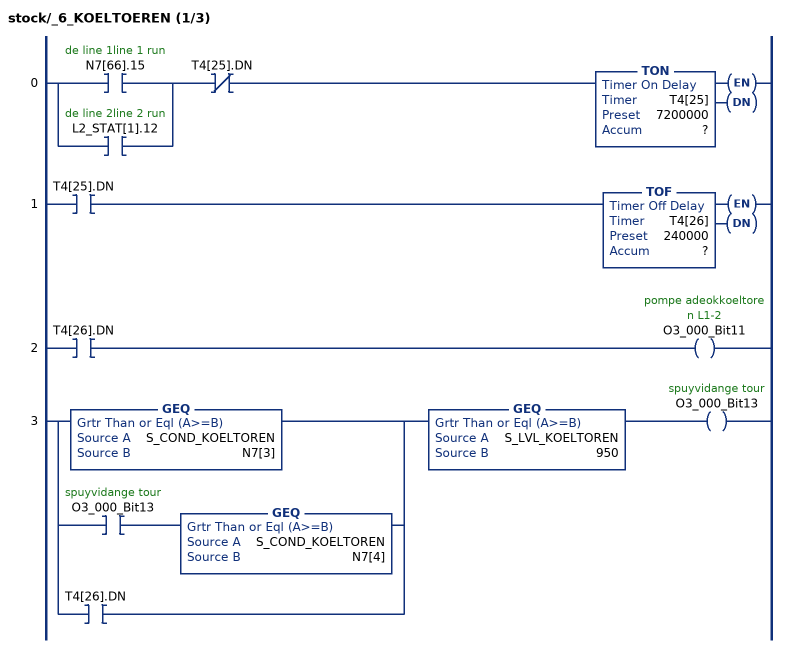
   0: [XIC(N7[66].15) ,XIC(L2_STAT[1].12) ]XIO(T4[25].DN)TON(T4[25],?,?);
   1: XIC(T4[25].DN)TOF(T4[26],?,?);
   2: XIC(T4[26].DN)OTE(O3_000_Bit11);
   3: [GEQ(S_COND_KOELTOREN,N7[3]) ,XIC(O3_000_Bit13) GEQ(S_COND_KOELTOREN,N7[4]) ,XIC(T4[26].DN) ]GEQ(S_LVL_KOELTOREN,950)OTE(O3_000_Bit13);
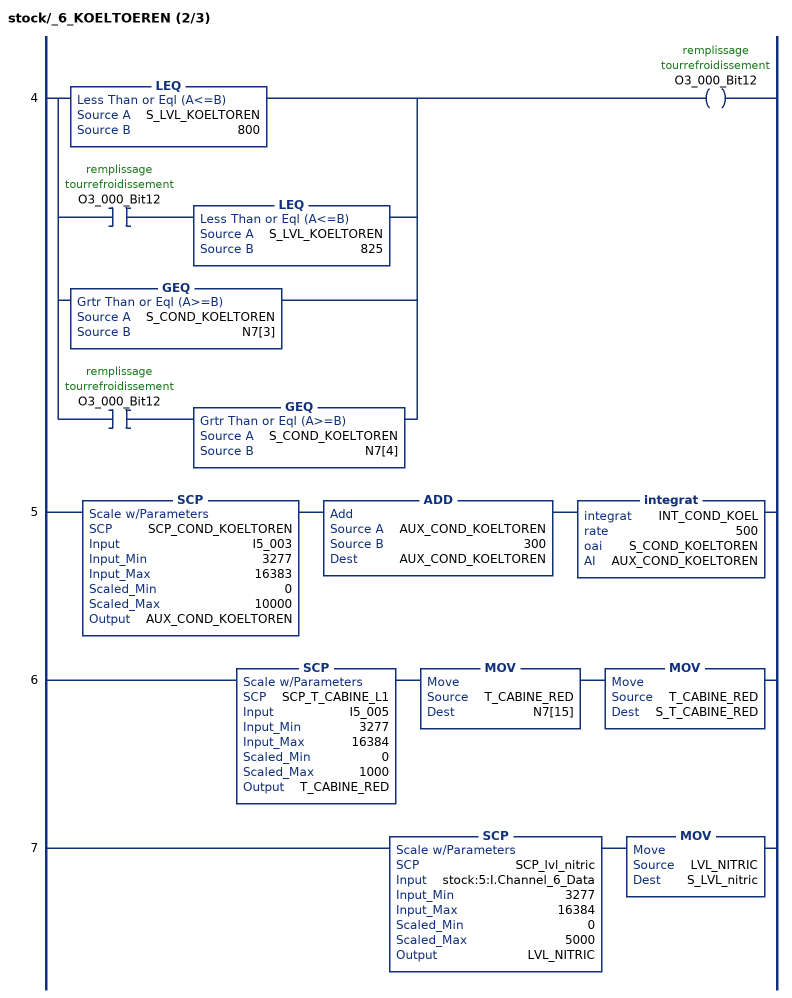
   4: [LEQ(S_LVL_KOELTOREN,800) ,XIC(O3_000_Bit12) LEQ(S_LVL_KOELTOREN,825) ,GEQ(S_COND_KOELTOREN,N7[3]) ,XIC(O3_000_Bit12) GEQ(S_COND_KOELTOREN,N7[4]) ]OTE(O3_000_Bit12);
   5: SCP(SCP_COND_KOELTOREN,I5_003,3277,16383,0,10000,AUX_COND_KOELTOREN)ADD(AUX_COND_KOELTOREN,300,AUX_COND_KOELTOREN)integrat(INT_COND_KOEL,500,S_COND_KOELTOREN,AUX_COND_KOELTOREN);
   6: SCP(SCP_T_CABINE_L1,I5_005,3277,16384,0,1000,T_CABINE_RED)MOV(T_CABINE_RED,N7[15])MOV(T_CABINE_RED,S_T_CABINE_RED);
   7: SCP(SCP_lvl_nitric,stock:5:I.Channel_6_Data,3277,16384,0,5000,LVL_NITRIC)MOV(LVL_NITRIC,S_LVL_nitric);
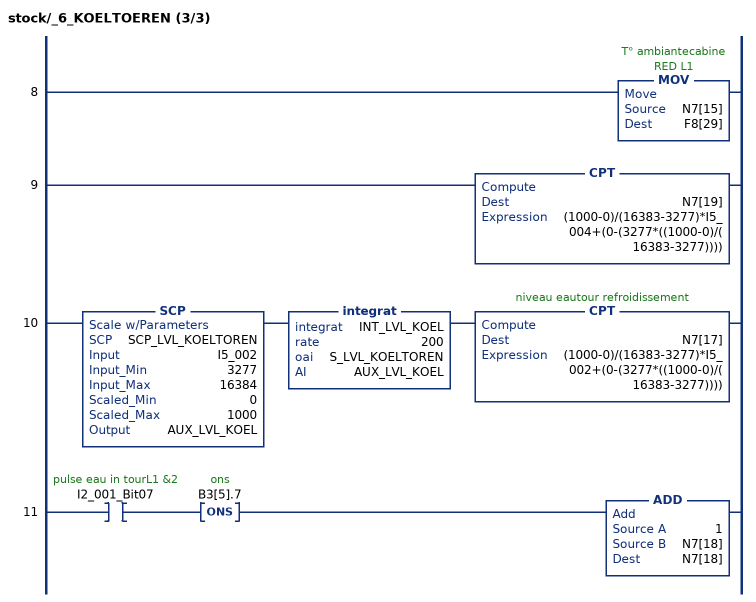
   8: MOV(N7[15],F8[29]);
   9: CPT(N7[19],(1000-0)/(16383-3277)*I5_004+(0-(3277*((1000-0)/(16383-3277)))));
   10: SCP(SCP_LVL_KOELTOREN,I5_002,3277,16384,0,1000,AUX_LVL_KOEL)integrat(INT_LVL_KOEL,200,S_LVL_KOELTOREN,AUX_LVL_KOEL)CPT(N7[17],(1000-0)/(16383-3277)*I5_002+(0-(3277*((1000-0)/(16383-3277)))));
   11: XIC(I2_001_Bit07)ONS(B3[5].7)ADD(1,N7[18],N7[18]);
END_ROUTINE

ROUTINE com   (* ladder *)
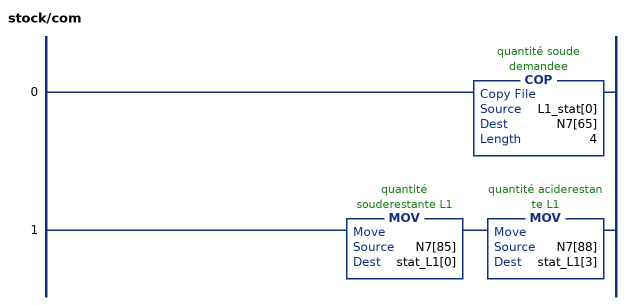
   0: COP(L1_stat[0],N7[65],4);
   1: MOV(N7[85],stat_L1[0])MOV(N7[88],stat_L1[3]);
END_ROUTINE

ROUTINE MAIN_STOCK   (* ladder *)
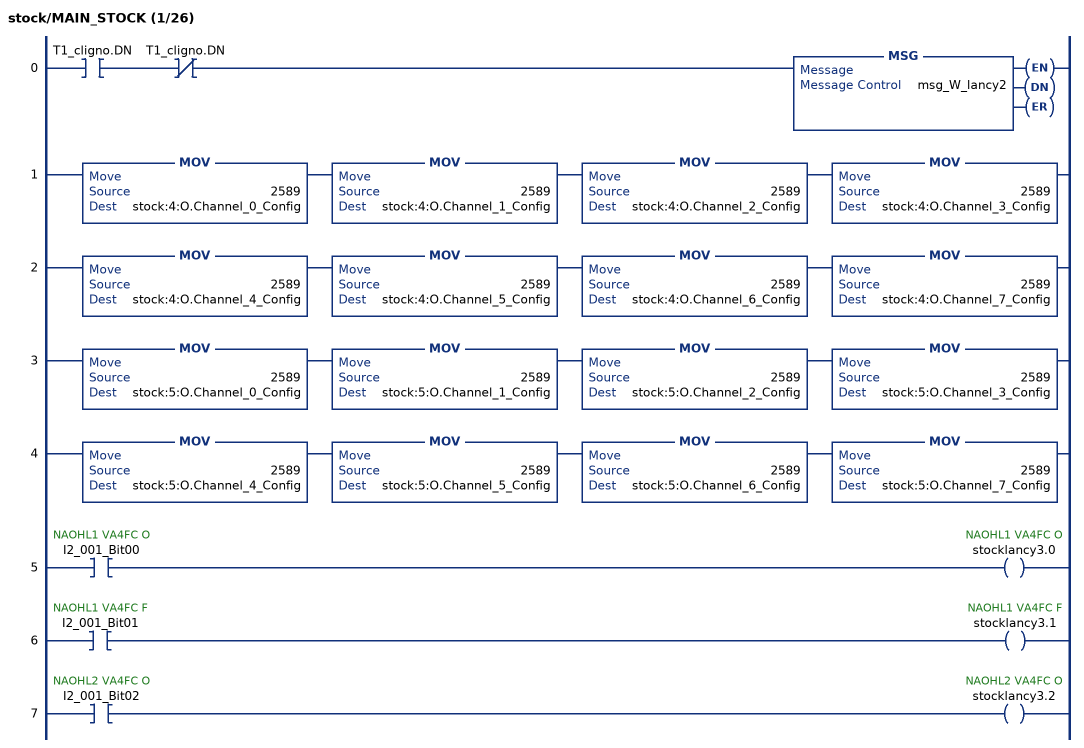
   0: XIC(T1_cligno.DN)XIO(T1_cligno.DN)MSG(msg_W_lancy2);
   1: MOV(2589,stock:4:O.Channel_0_Config)MOV(2589,stock:4:O.Channel_1_Config)MOV(2589,stock:4:O.Channel_2_Config)MOV(2589,stock:4:O.Channel_3_Config);
   2: MOV(2589,stock:4:O.Channel_4_Config)MOV(2589,stock:4:O.Channel_5_Config)MOV(2589,stock:4:O.Channel_6_Config)MOV(2589,stock:4:O.Channel_7_Config);
   3: MOV(2589,stock:5:O.Channel_0_Config)MOV(2589,stock:5:O.Channel_1_Config)MOV(2589,stock:5:O.Channel_2_Config)MOV(2589,stock:5:O.Channel_3_Config);
   4: MOV(2589,stock:5:O.Channel_4_Config)MOV(2589,stock:5:O.Channel_5_Config)MOV(2589,stock:5:O.Channel_6_Config)MOV(2589,stock:5:O.Channel_7_Config);
   5: XIC(I2_001_Bit00)OTE(stocklancy3.0);
   6: XIC(I2_001_Bit01)OTE(stocklancy3.1);
   7: XIC(I2_001_Bit02)OTE(stocklancy3.2);
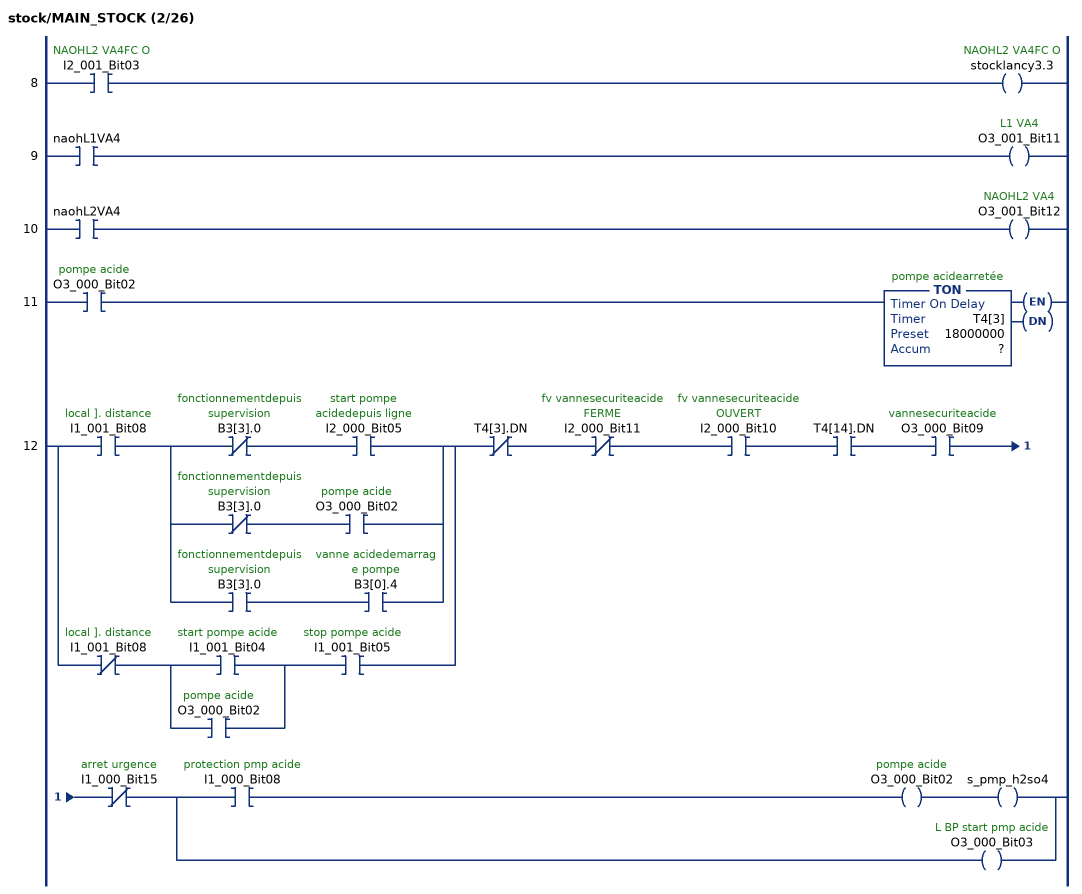
   8: XIC(I2_001_Bit03)OTE(stocklancy3.3);
   9: XIC(naohL1VA4)OTE(O3_001_Bit11);
   10: XIC(naohL2VA4)OTE(O3_001_Bit12);
   11: XIC(O3_000_Bit02)TON(T4[3],?,?);
   12: [XIC(I1_001_Bit08) [XIO(B3[3].0) XIC(I2_000_Bit05) ,XIO(B3[3].0) XIC(O3_000_Bit02) ,XIC(B3[3].0) XIC(B3[0].4) ] ,XIO(I1_001_Bit08) [XIC(I1_001_Bit04) ,XIC(O3_000_Bit02) ] XIC(I1_001_Bit05) ]XIO(T4[3].DN)XIO(I2_000_Bit11)XIC(I2_000_Bit10)XIC(T4[14].DN)XIC(O3_000_Bit09)XIO(I1_000_Bit15)[XIC(I1_000_Bit08) OTE(O3_000_Bit02) OTE(s_pmp_h2so4) ,OTE(O3_000_Bit03) ];
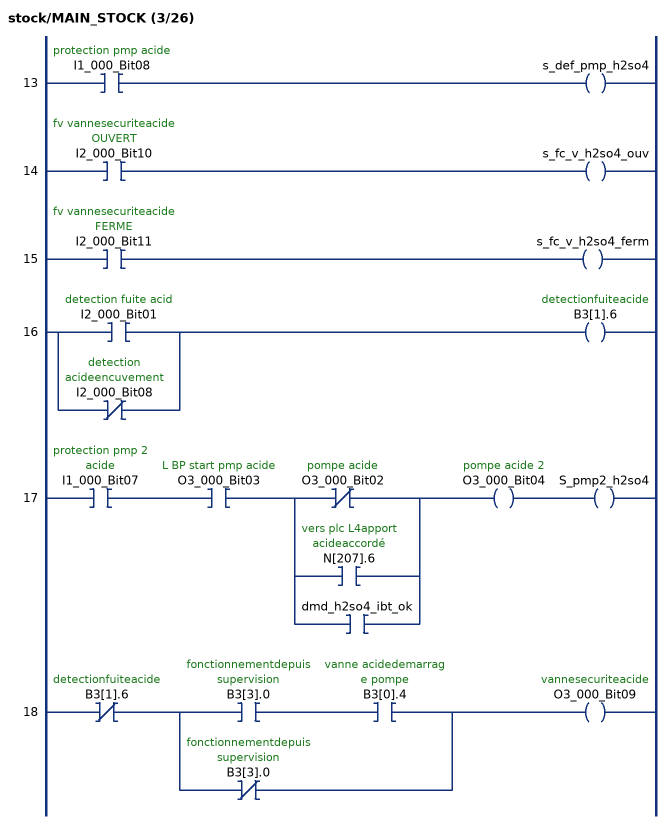
   13: XIC(I1_000_Bit08)OTE(s_def_pmp_h2so4);
   14: XIC(I2_000_Bit10)OTE(s_fc_v_h2so4_ouv);
   15: XIC(I2_000_Bit11)OTE(s_fc_v_h2so4_ferm);
   16: [XIC(I2_000_Bit01) ,XIO(I2_000_Bit08) ]OTE(B3[1].6);
   17: XIC(I1_000_Bit07)XIC(O3_000_Bit03)[XIO(O3_000_Bit02) ,XIC(N[207].6) ,XIC(dmd_h2so4_ibt_ok) ]OTE(O3_000_Bit04)OTE(S_pmp2_h2so4);
   18: XIO(B3[1].6)[XIC(B3[3].0) XIC(B3[0].4) ,XIO(B3[3].0) ]OTE(O3_000_Bit09);
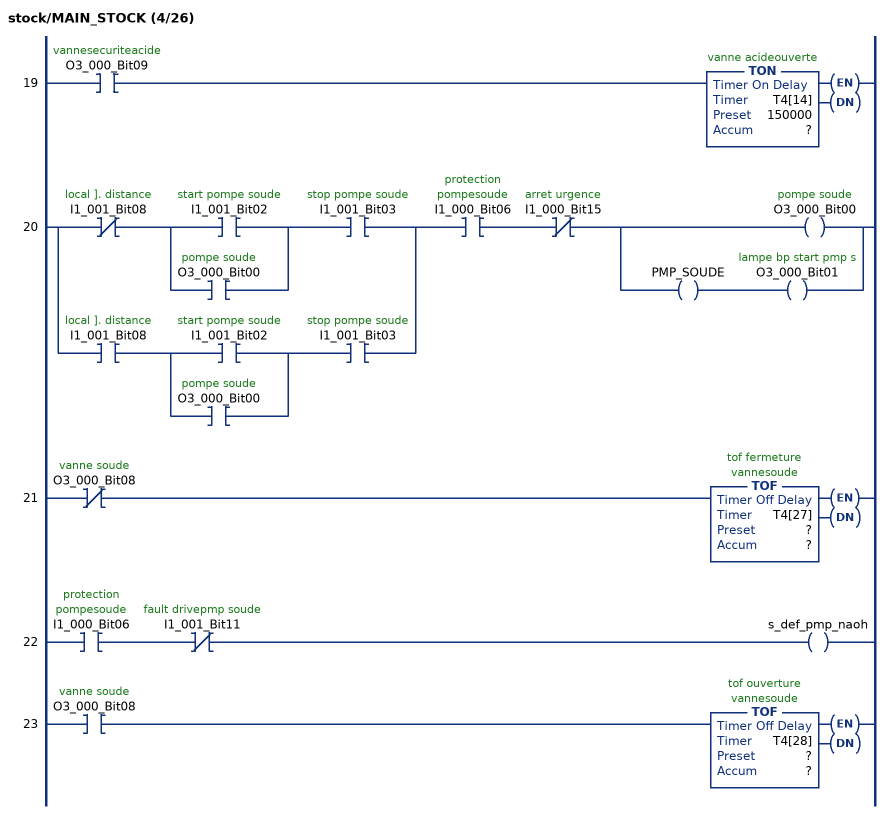
   19: XIC(O3_000_Bit09)TON(T4[14],?,?);
   20: [XIO(I1_001_Bit08) [XIC(I1_001_Bit02) ,XIC(O3_000_Bit00) ] XIC(I1_001_Bit03) ,XIC(I1_001_Bit08) [XIC(I1_001_Bit02) ,XIC(O3_000_Bit00) ] XIC(I1_001_Bit03) ]XIC(I1_000_Bit06)XIO(I1_000_Bit15)[OTE(O3_000_Bit00) ,OTE(PMP_SOUDE) OTE(O3_000_Bit01) ];
   21: XIO(O3_000_Bit08)TOF(T4[27],?,?);
   22: XIC(I1_000_Bit06)XIO(I1_001_Bit11)OTE(s_def_pmp_naoh);
   23: XIC(O3_000_Bit08)TOF(T4[28],?,?);
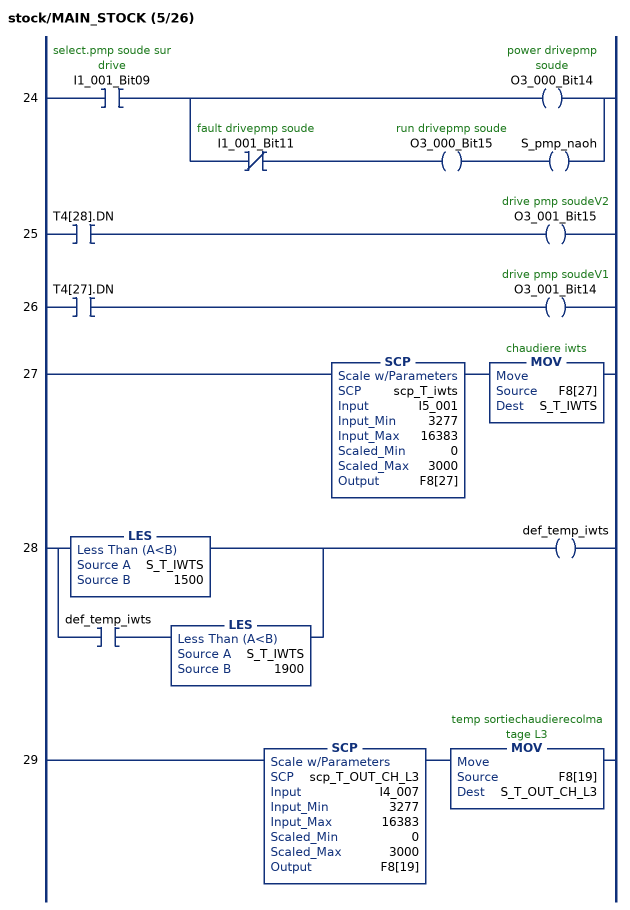
   24: XIC(I1_001_Bit09)[OTE(O3_000_Bit14) ,XIO(I1_001_Bit11) OTE(O3_000_Bit15) OTE(S_pmp_naoh) ];
   25: XIC(T4[28].DN)OTE(O3_001_Bit15);
   26: XIC(T4[27].DN)OTE(O3_001_Bit14);
   27: SCP(scp_T_iwts,I5_001,3277,16383,0,3000,F8[27])MOV(F8[27],S_T_IWTS);
   28: [LES(S_T_IWTS,1500) ,XIC(def_temp_iwts) LES(S_T_IWTS,1900) ]OTE(def_temp_iwts);
   29: SCP(scp_T_OUT_CH_L3,I4_007,3277,16383,0,3000,F8[19])MOV(F8[19],S_T_OUT_CH_L3);
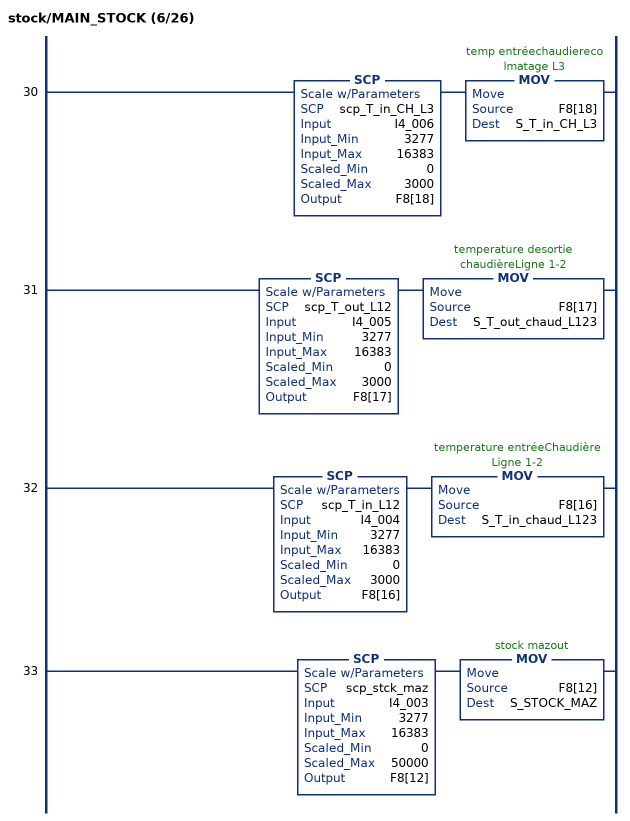
   30: SCP(scp_T_in_CH_L3,I4_006,3277,16383,0,3000,F8[18])MOV(F8[18],S_T_in_CH_L3);
   31: SCP(scp_T_out_L12,I4_005,3277,16383,0,3000,F8[17])MOV(F8[17],S_T_out_chaud_L123);
   32: SCP(scp_T_in_L12,I4_004,3277,16383,0,3000,F8[16])MOV(F8[16],S_T_in_chaud_L123);
   33: SCP(scp_stck_maz,I4_003,3277,16383,0,50000,F8[12])MOV(F8[12],S_STOCK_MAZ);
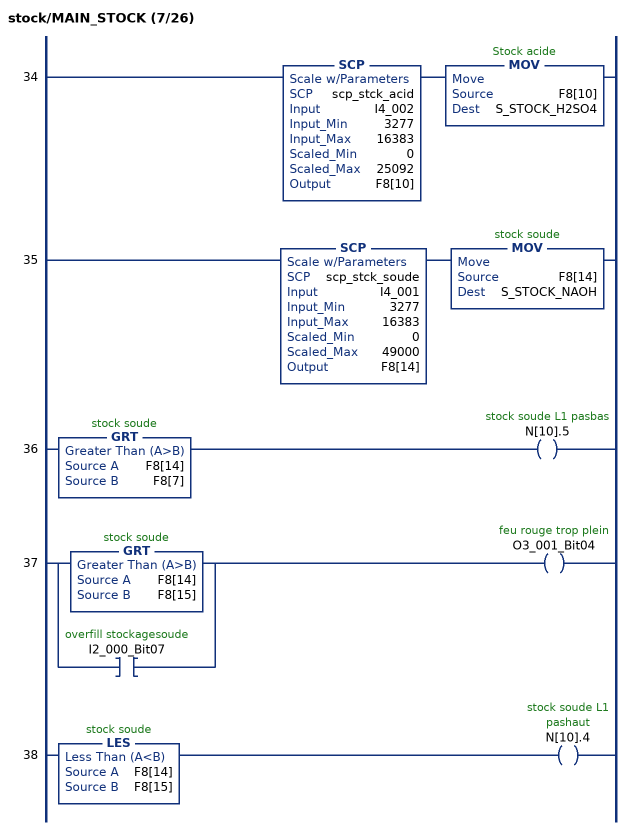
   34: SCP(scp_stck_acid,I4_002,3277,16383,0,25092,F8[10])MOV(F8[10],S_STOCK_H2SO4);
   35: SCP(scp_stck_soude,I4_001,3277,16383,0,49000,F8[14])MOV(F8[14],S_STOCK_NAOH);
   36: GRT(F8[14],F8[7])OTE(N[10].5);
   37: [GRT(F8[14],F8[15]) ,XIC(I2_000_Bit07) ]OTE(O3_001_Bit04);
   38: LES(F8[14],F8[15])OTE(N[10].4);
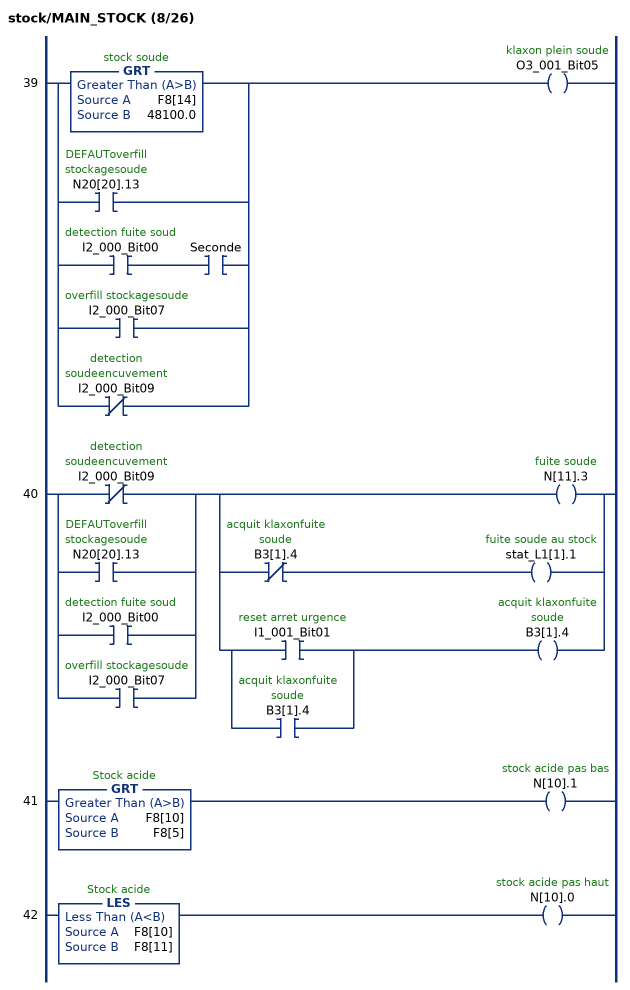
   39: [GRT(F8[14],48100.0) ,XIC(N20[20].13) ,XIC(I2_000_Bit00) XIC(Seconde) ,XIC(I2_000_Bit07) ,XIO(I2_000_Bit09) ]OTE(O3_001_Bit05);
   40: [XIO(I2_000_Bit09) ,XIC(N20[20].13) ,XIC(I2_000_Bit00) ,XIC(I2_000_Bit07) ][OTE(N[11].3) ,XIO(B3[1].4) OTE(stat_L1[1].1) ,[XIC(I1_001_Bit01) ,XIC(B3[1].4) ] OTE(B3[1].4) ];
   41: GRT(F8[10],F8[5])OTE(N[10].1);
   42: LES(F8[10],F8[11])OTE(N[10].0);
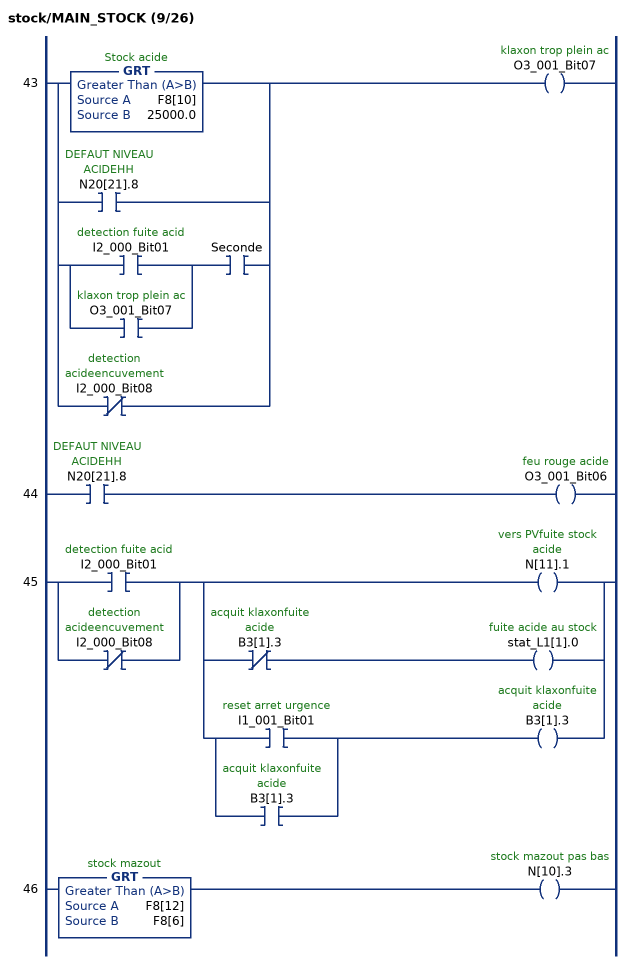
   43: [GRT(F8[10],25000.0) ,XIC(N20[21].8) ,[XIC(I2_000_Bit01) ,XIC(O3_001_Bit07) ] XIC(Seconde) ,XIO(I2_000_Bit08) ]OTE(O3_001_Bit07);
   44: XIC(N20[21].8)OTE(O3_001_Bit06);
   45: [XIC(I2_000_Bit01) ,XIO(I2_000_Bit08) ][OTE(N[11].1) ,XIO(B3[1].3) OTE(stat_L1[1].0) ,[XIC(I1_001_Bit01) ,XIC(B3[1].3) ] OTE(B3[1].3) ];
   46: GRT(F8[12],F8[6])OTE(N[10].3);
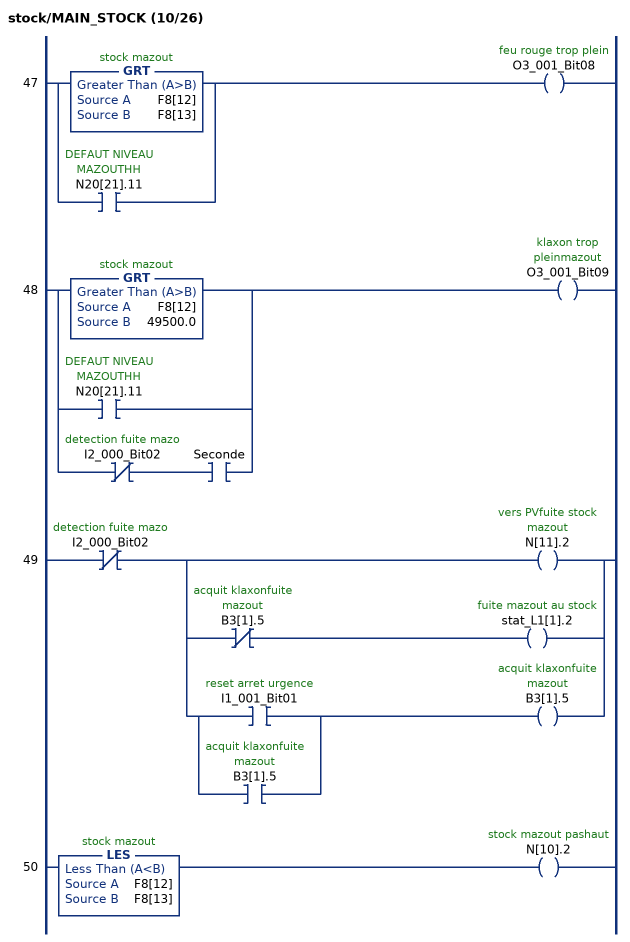
   47: [GRT(F8[12],F8[13]) ,XIC(N20[21].11) ]OTE(O3_001_Bit08);
   48: [GRT(F8[12],49500.0) ,XIC(N20[21].11) ,XIO(I2_000_Bit02) XIC(Seconde) ]OTE(O3_001_Bit09);
   49: XIO(I2_000_Bit02)[OTE(N[11].2) ,XIO(B3[1].5) OTE(stat_L1[1].2) ,[XIC(I1_001_Bit01) ,XIC(B3[1].5) ] OTE(B3[1].5) ];
   50: LES(F8[12],F8[13])OTE(N[10].2);
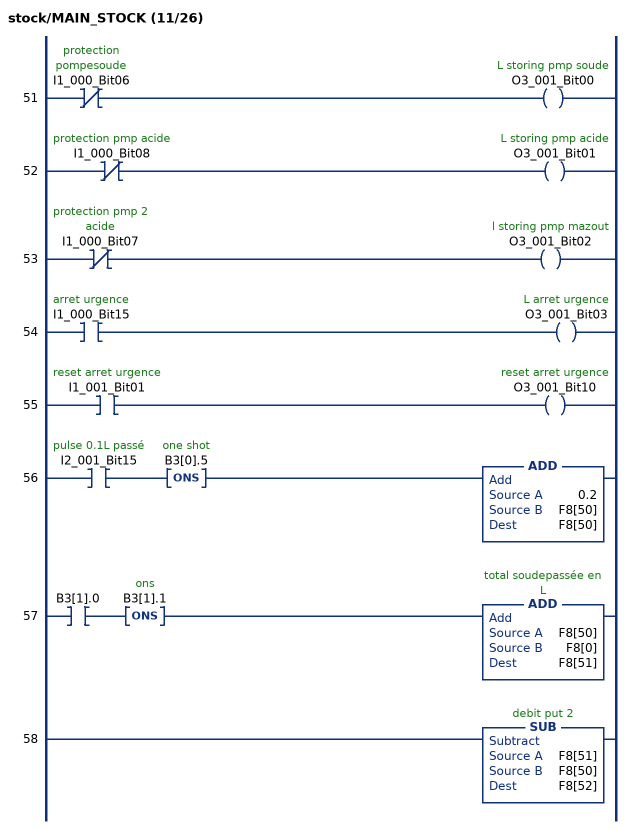
   51: XIO(I1_000_Bit06)OTE(O3_001_Bit00);
   52: XIO(I1_000_Bit08)OTE(O3_001_Bit01);
   53: XIO(I1_000_Bit07)OTE(O3_001_Bit02);
   54: XIC(I1_000_Bit15)OTE(O3_001_Bit03);
   55: XIC(I1_001_Bit01)OTE(O3_001_Bit10);
   56: XIC(I2_001_Bit15)ONS(B3[0].5)ADD(0.2,F8[50],F8[50]);
   57: XIC(B3[1].0)ONS(B3[1].1)ADD(F8[50],F8[0],F8[51]);
   58: SUB(F8[51],F8[50],F8[52]);
